// TIA Portal V17 export
// export: Created 2023-12-22T15:04:40.560973Z, ExportSetting WithDefaults, DisplayName Totally Integrated Automation Portal, DisplayVersion V17, DisplayName TIA Portal Openness, DisplayVersion V17, DisplayName TIA Portal Version Control Interface, DisplayVersion V17, DisplayName STEP 7 Professional, DisplayVersion V17, DisplayName STEP 7 Safety, DisplayVersion V17, DisplayName WinCC Advanced, DisplayVersion V17
FUNCTION_BLOCK "DO_ex"   // FB102, LAD
{ S7_Optimized_Access := 'FALSE' }
VERSION : 0.1
// stored: AutoNumber false, IsIECCheckEnabled false, SetENOAutomatically false, UDAEnableTagReadback false
   VAR_INPUT
      REQ : Bool;   // Запрос включения
      All_Block : Bool;
   END_VAR
   VAR_IN_OUT
      Q : Bool;   // Выходной сигнал ПЛК
   END_VAR
   VAR DB_SPECIFIC
      CMD : "CMD";   // Основные команды / Блок команд
      Use : Struct   // Функционал
         Inverse { S7_SetPoint := 'True'} : Bool;   // Инверсия входного сигнала
         Indirect { S7_SetPoint := 'True'} : Bool := true;   // Использование косвенной адресации
         Impulse { S7_SetPoint := 'True'} : Bool;   // Использовать импульсный режим
      END_STRUCT;
      ADDR_Byte { S7_SetPoint := 'True'} : Int;   // Адрес входа на контроллере (Байт)
      ADDR_Bit { S7_SetPoint := 'True'} : Int := 9;   // Адрес входа на контроллере (Бит)
      Mode : Int;
      Status : Int;
   END_VAR
   VAR
      T_Impulse { S7_SetPoint := 'True'} : "Time_S_b";   // Длительность импульса
   END_VAR
   VAR_TEMP
      Start : Bool;
   END_VAR
   VAR_TEMP   // added for the SCL form of the ladder/FBD networks
      _w1 : Bool;
   END_VAR
BEGIN

REGION Network 1: Устройство в ручном режиме
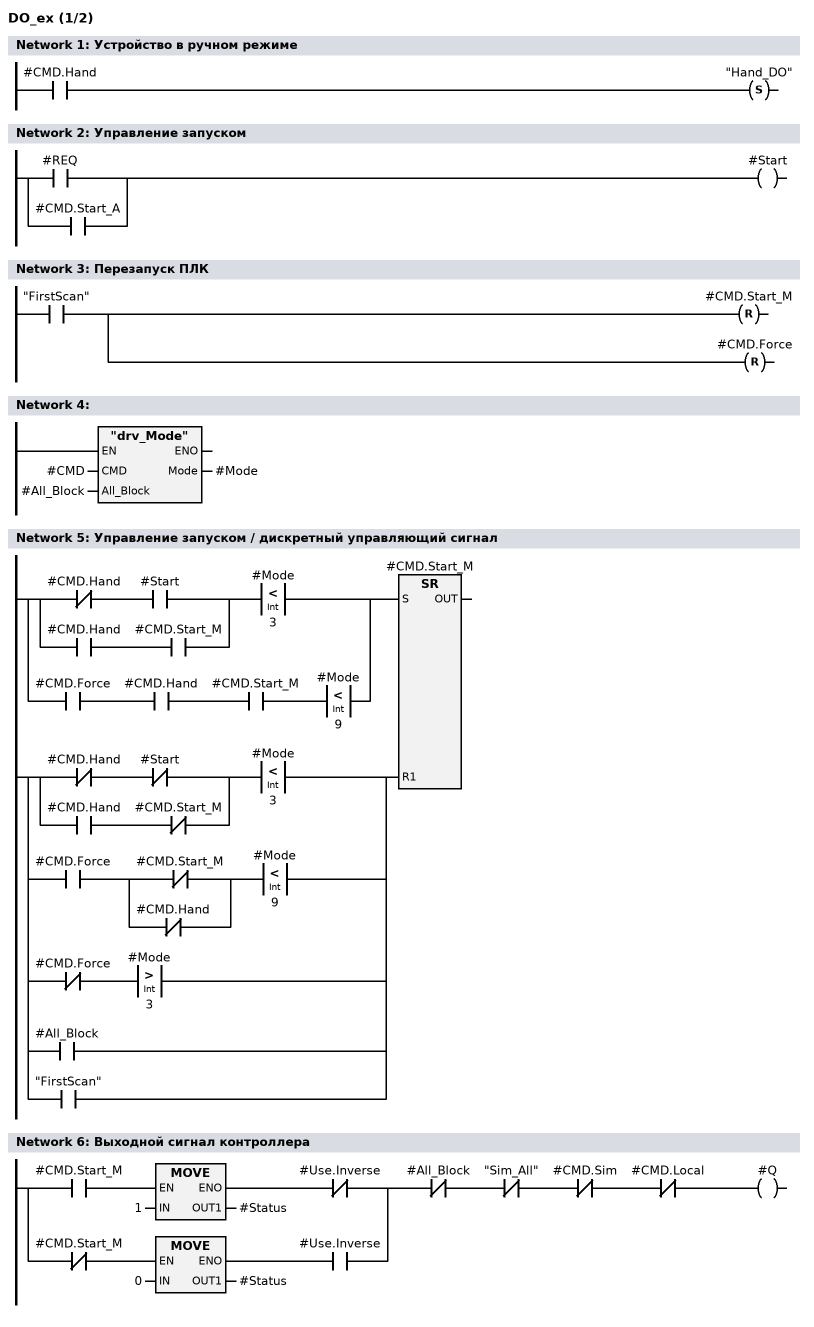
   RUNG wire#powerrail
      Contact( #CMD.Hand )
      S_Coil( "Hand_DO" )
   END_RUNG
   // the same network as SCL:
   IF #CMD.Hand THEN "Hand_DO" := TRUE; END_IF;
END_REGION

REGION Network 2: Управление запуском
   RUNG wire#powerrail
      Contact( #REQ )
      wire#w1
      Coil( #Start )
   END_RUNG
   RUNG wire#powerrail
      Contact( #CMD.Start_A )
   END_RUNG wire#w1
   // the same network as SCL:
   #Start := #REQ OR #CMD.Start_A;
END_REGION

REGION Network 3: Перезапуск ПЛК
   RUNG wire#powerrail
      Contact( "FirstScan" )
      wire#w1
      R_Coil( #CMD.Start_M )
   END_RUNG
   RUNG wire#w1
      R_Coil( #CMD.Force )
   END_RUNG
   // the same network as SCL:
   IF "FirstScan" THEN
       #CMD.Start_M := FALSE;
       #CMD.Force := FALSE;
   END_IF;
END_REGION

REGION Network 4
   RUNG wire#powerrail
      "drv_Mode"(CMD := #CMD, All_Block := #All_Block, Mode => #Mode)
   END_RUNG
   // the same network as SCL:
   "drv_Mode"(CMD := #CMD, All_Block := #All_Block, Mode => #Mode);
END_REGION

REGION Network 5: Управление запуском / дискретный управляющий сигнал
   RUNG wire#powerrail
      I_Contact( #CMD.Hand )
      Contact( #Start )
      wire#w1
      { S7_Templates := "SrcType := Int" } LT_Contact(in1 := #Mode, in2 := 3)
      wire#w2
      S_SR(operand := #CMD.Start_M, r1 := wire#w6)
   END_RUNG
   RUNG wire#powerrail
      Contact( #CMD.Hand )
      Contact( #CMD.Start_M )
   END_RUNG wire#w1
   RUNG wire#powerrail
      Contact( #CMD.Force )
      Contact( #CMD.Hand )
      Contact( #CMD.Start_M )
      { S7_Templates := "SrcType := Int" } LT_Contact(in1 := #Mode, in2 := 9)
   END_RUNG wire#w2
   RUNG wire#powerrail
      I_Contact( #CMD.Hand )
      I_Contact( #Start )
      wire#w3
      { S7_Templates := "SrcType := Int" } LT_Contact(in1 := #Mode, in2 := 3)
   END_RUNG wire#w6
   RUNG wire#powerrail
      Contact( #CMD.Hand )
      I_Contact( #CMD.Start_M )
   END_RUNG wire#w3
   RUNG wire#powerrail
      Contact( #CMD.Force )
      wire#w4
      I_Contact( #CMD.Start_M )
      wire#w5
      { S7_Templates := "SrcType := Int" } LT_Contact(in1 := #Mode, in2 := 9)
   END_RUNG wire#w6
   RUNG wire#w4
      I_Contact( #CMD.Hand )
   END_RUNG wire#w5
   RUNG wire#powerrail
      I_Contact( #CMD.Force )
      { S7_Templates := "SrcType := Int" } GT_Contact(in1 := #Mode, in2 := 3)
   END_RUNG wire#w6
   RUNG wire#powerrail
      Contact( #All_Block )
   END_RUNG wire#w6
   RUNG wire#powerrail
      Contact( "FirstScan" )
   END_RUNG wire#w6
   // the same network as SCL:
   #_w1 := (((NOT #CMD.Hand AND NOT #Start) OR (#CMD.Hand AND NOT #CMD.Start_M)) AND (#Mode < 3)) OR (#CMD.Force AND (NOT #CMD.Start_M OR NOT #CMD.Hand) AND (#Mode < 9)) OR (NOT #CMD.Force AND (#Mode > 3)) OR #All_Block OR "FirstScan";
   IF (((NOT #CMD.Hand AND #Start) OR (#CMD.Hand AND #CMD.Start_M)) AND (#Mode < 3)) OR (#CMD.Force AND #CMD.Hand AND #CMD.Start_M AND (#Mode < 9)) THEN
       #CMD.Start_M := TRUE;   // SR flip-flop
   END_IF;
   IF #_w1 THEN #CMD.Start_M := FALSE; END_IF;
END_REGION

REGION Network 6: Выходной сигнал контроллера
   RUNG wire#powerrail
      Contact( #CMD.Start_M )
      Move(in := 1, out1 => #Status)
      I_Contact( #Use.Inverse )
      wire#w1
      I_Contact( #All_Block )
      I_Contact( "Sim_All" )
      I_Contact( #CMD.Sim )
      I_Contact( #CMD.Local )
      Coil( #Q )
   END_RUNG
   RUNG wire#powerrail
      I_Contact( #CMD.Start_M )
      Move(in := 0, out1 => #Status)
      Contact( #Use.Inverse )
   END_RUNG wire#w1
   // the same network as SCL:
   IF #CMD.Start_M THEN #Status := 1; END_IF;
   IF NOT #CMD.Start_M THEN #Status := 0; END_IF;
   #Q := ((#CMD.Start_M AND NOT #Use.Inverse) OR (NOT #CMD.Start_M AND #Use.Inverse)) AND NOT #All_Block AND NOT "Sim_All" AND NOT #CMD.Sim AND NOT #CMD.Local;
END_REGION

REGION Network 7: Косвенная адресация
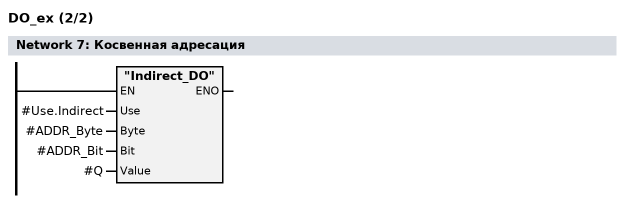
   RUNG wire#powerrail
      "Indirect_DO"(Use := #Use.Indirect, "Byte" := #ADDR_Byte, Bit := #ADDR_Bit, Value := #Q)
   END_RUNG
   // the same network as SCL:
   "Indirect_DO"(Use := #Use.Indirect, "Byte" := #ADDR_Byte, Bit := #ADDR_Bit, Value := #Q);
END_REGION
END_FUNCTION_BLOCK
